// TIA Portal project "Traffic_feuxFBD" (V15)

(* hardware
DEVICE "Station S7300/ET200M_1"  S7-300 station
   slot 0: "Châssis_0"  Rail  6ES7 390-1***0-0AA0
   slot 2: "PLC_1"  CPU 315-2 PN/DP  6ES7 315-2EH14-0AB0  V3.2
      slot 2: "Interface PROFINET_1"  PN-IO
         slot 1: "Port_1"  Port
         slot 2: "Port_2"  Port
DEVICE "HMI_1"  KTP900 Basic PN
   slot 0: "HMI_1"  KTP900 Basic PN  6AV2 123-2JB03-0AX0  15.0.0.0
   slot 1: "HMI_RT_1"  KTP900 Basic PN  6AV2 123-2JB03-0AX0  15.0.0.0
   slot 5: "HMI_1.IE_CP_1"  PROFINET Interface  15.0.0.0
      slot 1: "Interface PROFINET_1"  PROFINET Interface
         slot 1: "Port_1"  Port
*)

// ===== PLC "PLC_1"  CPU 315-2 PN/DP =====

VAR_GLOBAL   // PLC tag table "Light_table"
   "Lred" AT %Q0.0 : Bool;
   "Lgreen" AT %Q0.1 : Bool;
   "Lorange" AT %Q0.2 : Bool;
   "Start" AT %I0.0 : Bool;
END_VAR

DATA_BLOCK "Bloc_1_DB"   // DB1
{ S7_Optimized_Access := 'FALSE' }
VERSION : 0.1
// stored: InstanceOfName Bloc_1
"Bloc_1"
BEGIN
END_DATA_BLOCK

FUNCTION_BLOCK "Bloc_1"   // FB1, GRAPH
{ S7_Optimized_Access := 'FALSE' }
VERSION : 0.1
   VAR_INPUT
      OFF_SQ : Bool := false;   // Désactiver le graphe
      INIT_SQ : Bool := false;   // Mettre le graphe à l'état initial
      ACK_EF : Bool := false;   // Acquitter toutes les erreurs et perturbations
      S_PREV : Bool := false;   // Afficher l'étape précédente dans le paramètre S_NO
      S_NEXT : Bool := false;   // Afficher l'étape suivante dans le paramètre S_NO
      SW_AUTO : Bool := false;   // Mode automatique
      SW_TAP : Bool := false;   // Mode semi-automatique/Activation de l'étape suivante avec transition
      SW_TOP : Bool := false;   // Mode semi-automatique/Ignorer la transition
      SW_MAN : Bool := false;   // Mode manuel
      S_SEL : Int := 0;   // Sélectionner l'étape à afficher dans S_NO
      S_ON : Bool := false;   // Activer l'étape figurant dans le paramètre S_NO
      S_OFF : Bool := false;   // Désactiver l'étape figurant dans le paramètre S_NO
      T_PUSH : Bool := false;   // Validation de commutation pour transition en mode semi-automatique
   END_VAR
   VAR_OUTPUT
      S_NO : Int := 0;   // Numéro d'étape
      S_MORE : Bool := false;   // Il existe d'autres étapes qui peuvent être affichées dans S_NO.
      S_ACTIVE : Bool := false;   // L'étape affichée dans le paramètre S_NO est activée
      ERR_FLT : Bool := false;   // Erreur groupée Interlock or Supervision
      AUTO_ON : Bool := false;   // Mode automatique activé
      TAP_ON : Bool := false;   // Mode semi-automatique/Etape avec transition activé
      TOP_ON : Bool := false;   // Mode semi-automatique/Ignorer la transition activé
      MAN_ON : Bool := false;   // Mode manuel activé
   END_VAR
   VAR
      SWITCH : Array[0..0] of DWord;
      SW_SQTS : Array[0..3] of Byte;
      SW_ADDR : Word := 16#A;
      G7T_0 : GraphTransition;
      G7S_0 : GraphStep;
      PRE_CRIT : Array[0..0] of DWord;
      POST_CRIT : Array[0..0] of DWord;
      TVX : Array[0..2] of Byte;
      TTX : Array[0..2] of Byte;
      TSX : Array[0..2] of Byte;
      S00X : Array[0..2] of Byte;
      SOFFX : Array[0..2] of Byte;
      SONX : Array[0..2] of Byte;
      SAX : Array[0..2] of Byte;
      SERRX : Array[0..4] of Byte;
      SMX : Array[0..4] of Byte;
      S0X : Array[0..4] of Byte;
      S1X : Array[0..4] of Byte;
      S_DISPLAY : Int;   // Affichage interne du paramètre de sortie S_NO
      S_SEL_OLD : Int;   // Valeur précédente dans S_SEL
      S_DISPIDX : Byte;   // Indice de l'étape affichée dans S_NO
      T_DISPIDX : Byte;   // Indice de la transition affichée dans T_NO
      MOPEDGE : Struct
         AUTO : Bool := false;
         MAN : Bool := false;
         TAP : Bool := false;
         TOP : Bool := false;
         ACK_S : Bool := false;
         REG_S : Bool := false;
         T_PREV : Bool := false;
         T_NEXT : Bool := false;
         LOCK : Bool := false;
         SUP : Bool := false;
         ACKREQ : Bool := false;
         SSKIP : Bool := false;
         OFF : Bool := false;
         INIT : Bool := false;
         HALT : Bool := false;
         TMS_HALT : Bool := false;
         OPS_ZERO : Bool := false;
         SACT_DISP : Bool := false;
         SEF_DISP : Bool := false;
         SALL_DISP : Bool := false;
         S_PREV : Bool := false;
         S_NEXT : Bool := false;
         S_SELOK : Bool := false;
         S_ON : Bool := false;
         S_OFF : Bool := false;
         T_PUSH : Bool := false;
         REG : Bool := false;
         ACK : Bool := false;
         IL_PERM : Bool := false;
         T_PERM : Bool := false;
         ILP_MAN : Bool := false;
      END_STRUCT;
      MOP : Struct   // Mode de fonctionnement
         AUTO : Bool := true;   // Etat : Mode automatique
         MAN : Bool := false;   // Etat : Mode manuel
         TAP : Bool := false;   // Etat : Mode semi-automatique/Activation de l'étape suivante avec transition
         TOP : Bool := false;   // Etat : Mode semi-automatique/Ignorer la transition
         ACK_S : Bool := false;   // Requête : Acquitter l'étape figurant dans le paramètre S_NO
         REG_S : Bool := false;   // Requête : Enregistrer l'étape figurant dans le paramètre S_NO
         T_PREV : Bool := false;   // Requête : Afficher la transition valide précédente dans le paramètre T_NO
         T_NEXT : Bool := false;   // Requête : Afficher la transition valide suivante dans le paramètre T_NO
         LOCK : Bool := true;   // Etat : Traitement des Interlocks activé
         SUP : Bool := true;   // Etat : Traitement de Supervision activé
         ACKREQ : Bool := true;   // Etat : Acquittement requis
         SSKIP : Bool := false;   // Etat : "Ignorer les étapes" activé
         OFF : Bool := false;   // Requête : Désactiver toutes les étapes
         INIT : Bool := true;   // Requête : Mettre le graphe à l'état initial
         HALT : Bool := false;   // Etat : Le graphe est arrêté
         TMS_HALT : Bool := false;   // Etat : Toutes les temporisations internes sont arrêtées
         OPS_ZERO : Bool := false;   // Etat : Tous les opérandes traités avec N, L, D mis à 0
         SACT_DISP : Bool := true;   // Etat : N'afficher que les étapes actives
         SEF_DISP : Bool := false;   // Etat : Afficher uniquement les étapes avec erreurs et perturbations
         SALL_DISP : Bool := false;   // Etat : Afficher toutes les étapes
         S_PREV : Bool := false;   // Requête : Afficher l'étape précédente dans le paramètre S_NO
         S_NEXT : Bool := false;   // Requête : Afficher l'étape suivante dans le paramètre S_NO
         S_SELOK : Bool := false;   // Requête : Afficher dans le paramètre S_NO le numéro d'étape figurant dans S_SEL
         S_ON : Bool := false;   // Requête : Activer l'étape figurant dans le paramètre S_NO
         S_OFF : Bool := false;   // Requête : Désactiver l'étape figurant dans le paramètre S_NO
         T_PUSH : Bool := false;   // Requête : Validation de commutation pour transition
         REG : Bool := false;   // Requête : Enregistrer toutes les erreurs Interlock et Supervision
         ACK : Bool := false;   // Requête : Acquitter toutes les erreurs Interlock et Supervision
         IL_PERM : Bool := false;   // Etat : Traitement permanent de tous les Interlocks
         T_PERM : Bool := false;   // Etat : Traitement permanent de toutes les transitions
         ILP_MAN : Bool := false;   // Etat : Traitement permanent de tous les Interlocks en mode manuel
      END_STRUCT;
      TICKS : Struct   // Périodes d'horloge
         DELTA : Time := T#0ms;   // Différence de temps entre deux cycles
         OLD : Time := T#0ms;   // Valeur du compteur de périodes 10 ms au dernier cycle
         NEW : Time := T#0ms;   // Valeur du compteur de périodes 10 ms dans ce cycle
      END_STRUCT;
      SQ_FLAGS : Struct   // Mémentos de graphe
         ERR_FLT : Bool := false;   // Erreur groupée Interlock et Supervision
         ERROR : Bool := false;   // Erreur groupée Interlock
         FAULT : Bool := false;   // Erreur groupée Supervision
         RT_FAIL : Bool := false;   // Erreur à l'exécution
         NO_SNO : Bool := false;   // Numéro d'étape requis introuvable
         NF_OFL : Bool := false;   // Débordement : Trop de requêtes ON ou OFF
         SA_OFL : Bool := false;   // Débordement : Trop d'étapes activées
         TV_OFL : Bool := false;   // Débordement : Trop de transitions valides
         MSG_OFL : Bool := false;   // Débordement : Pas assez de ressources système pour ALARM_S
         NO_SWI : Bool := false;   // Pas de commutation dans ce cycle
         CYC_OP : Bool := false;   // Exécution cyclique du graphe après l'initialisation
         AS_MSG : Bool := true;   // Messages à l'exécution activés ou désactivés par instruction
         AS_SEND : Bool := false;   // Envoyer les messages de WR_USMSG ou les entrer uniquement dans le tampon de diagnostic
         SQ_BUSY : Bool := false;   // Mémento de front interne pour le traitement séquentiel
         SA_BUSY : Bool := false;   // Mémento de front interne pour le traitement séquentiel
         AS_SIG : Bool := false;   // Mémentos de front pour messages de Alarm_S et Alarm_SQ
      END_STRUCT;
      S_PTR : DWord := 16#2A0;
      S_PTR2 : DWord := 16#0;
      S_PTR3 : DWord := 16#850;
      S_PTR4 : DWord := 16#820;
      T_PTR : DWord := 16#7F0;
      C_AR2 : DWord := 16#0;
      M_FBDB : DWord := 16#10000;
      M_SNO : Word := 16#0;
      M_EVID : Word := 16#0;
      M_EVIL : C_Alarm_s;
      M_EVSV : C_Alarm_s;
      M_EV : DWord := 16#760;
      CRIT : Array[0..31] of Bool;
      S_START : Byte := 16#0;
      S_IDX : Byte := 16#0;
      S_INT : Int := 72;
      S_TMP : Byte := 16#0;
      T_START : Byte := 16#0;
      T_IDX : Byte := 16#0;
      T_TMP : Byte := 16#0;
      T_TMP2 : Byte := 16#00;
      TV_POT : Byte := 16#06;
      RETURN1 : Byte := 16#0;
      RETURN2 : Byte := 16#0;
      SINI : Array[0..2] of Byte;
      LSTT : Array[0..3] of Byte;
      ATAJ : Array[0..3] of Byte;
      ATAB : Array[0..3] of Byte;
      PSTT : Array[0..3] of Byte;
      NSTT : Array[0..3] of Byte;
      ASSJ : Array[0..3] of Byte;
      ASSB : Array[0..3] of Byte;
      PTTS : Array[0..3] of Byte;
      NTTS : Array[0..3] of Byte;
      PRE_CNT : Word := 16#1;
      POST_CNT : Word := 16#1;
      ADR_COND : Word := 16#0;
      MAX_TVAL : Byte := 16#1;
      MAX_SACT : Byte := 16#1;
      MAX_CRIT : Byte := 16#4;
      T_CNT : Byte := 16#3;
      SUP_CNT : Byte := 16#0;
      LOCK_CNT : Byte := 16#0;
      S_CNT : Byte := 16#3;
      SQ_CNT : Byte := 16#1;
      PRS_INPAR : DWord := 16#E000FEC8;
      PRS_OUTPAR : DWord := 16#E000800F;
      GC_FLAGS : Struct
         T_MACH : Byte := 16#EB;
         COND_ED : Byte := 16#E3;
         W_LEVEL : Byte := 16#D5;
         FB_IF : Byte := 16#FA;
         AS_MSG : Word := 16#404;
         SSB : Word := 16#108;
         DILG : Word := 16#1B8;
         ADDR_T0 : Word := 16#14;
         CRIT_AVAIL : Bool := false;
         SSKIP_AVAIL : Bool := true;
         SSKIP_ON : Bool := false;
         ACK_REQ : Bool := true;
         SYNC_AVAIL : Bool := true;
         ILP_MAN : Bool := false;
         SWM_LOCKED : Bool := false;
         SAVE_SW : Bool := true;
      END_STRUCT;
      G7_FBMARK : Byte := 16#3C;
      G7_RELEASE : Byte := 16#3C;
      G7_ID2 : Byte := 16#37;
      G7_ID1 : Byte := 16#47;
   END_VAR
   // SW_SQTS[0] := 16#1;
   // TVX[0] := 16#1;
   // TTX[0] := 16#1;
   // TSX[0] := 16#1;
   // S00X[0] := 16#1;
   // SOFFX[0] := 16#1;
   // SONX[0] := 16#1;
   // SAX[0] := 16#1;
   // SERRX[0] := 16#1;
   // SMX[0] := 16#1;
   // S0X[0] := 16#1;
   // S1X[0] := 16#1;
   // SINI[0] := 16#2;
   // SINI[1] := 16#1;
   // SINI[2] := 0;
   // LSTT[0] := 0;
   // LSTT[1] := 0;
   // LSTT[2] := 0;
   // LSTT[3] := 16#1;
   // ATAJ[0] := 0;
   // ATAJ[1] := 16#1;
   // ATAJ[2] := 16#2;
   // ATAJ[3] := 16#3;
   // ATAB[0] := 0;
   // ATAB[1] := 16#1;
   // ATAB[2] := 16#2;
   // ATAB[3] := 16#3;
   // PSTT[0] := 0;
   // PSTT[1] := 16#1;
   // PSTT[2] := 16#2;
   // PSTT[3] := 16#3;
   // NSTT[0] := 16#1;
   // NSTT[1] := 16#2;
   // NSTT[2] := 16#3;
   // NSTT[3] := 16#1;
   // ASSJ[0] := 0;
   // ASSJ[1] := 16#1;
   // ASSJ[2] := 16#2;
   // ASSJ[3] := 16#3;
   // ASSB[0] := 0;
   // ASSB[1] := 16#1;
   // ASSB[2] := 16#2;
   // ASSB[3] := 16#3;
   // PTTS[0] := 0;
   // PTTS[2] := 16#1;
   // PTTS[3] := 16#2;
   // NTTS[0] := 0;
   // NTTS[1] := 16#1;
   // NTTS[2] := 16#2;
   // NTTS[3] := 16#3;
BEGIN
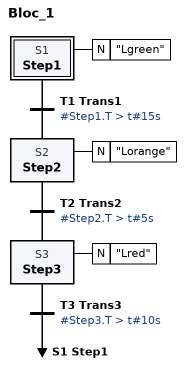
   // sequencer 1
   INITIAL_STEP Step1:   // S1
              N    "Lgreen"
   END_STEP
   TRANSITION Trans1 FROM Step1 TO Step2   // T1
      := #Step1.T > t#15s;
   END_TRANSITION
   STEP Step2:   // S2
              N    "Lorange"
   END_STEP
   TRANSITION Trans2 FROM Step2 TO Step3   // T2
      := #Step2.T > t#5s;
   END_TRANSITION
   STEP Step3:   // S3
              N    "Lred"
   END_STEP
   TRANSITION Trans3 FROM Step3 TO Step1   // T3, jump
      := #Step3.T > t#10s;
   END_TRANSITION
END_FUNCTION_BLOCK

ORGANIZATION_BLOCK "Main"   // OB1, LAD
TITLE = "Main Program Sweep (Cycle)"
{ S7_Optimized_Access := 'FALSE' }
VERSION : 0.1
   VAR_TEMP
      OB1_EV_CLASS : Byte;   // Bits 0-3 = 1 (Coming event), Bits 4-7 = 1 (Event class 1)
      OB1_SCAN_1 : Byte;   // 1 (Cold restart scan 1 of OB 1), 3 (Scan 2-n of OB 1)
      OB1_PRIORITY : Byte;   // Priority of OB Execution
      OB1_OB_NUMBR : Byte;   // 1 (Organization block 1, OB1)
      OB1_RESERVED_1 : Byte;   // Reserved for system
      OB1_RESERVED_2 : Byte;   // Reserved for system
      OB1_PREV_CYCLE : Int;   // Cycle time of previous OB1 scan (milliseconds)
      OB1_MIN_CYCLE : Int;   // Minimum cycle time of OB1 (milliseconds)
      OB1_MAX_CYCLE : Int;   // Maximum cycle time of OB1 (milliseconds)
      OB1_DATE_TIME : Date_And_Time;   // Date and time OB1 started
   END_VAR
BEGIN

REGION Network 1
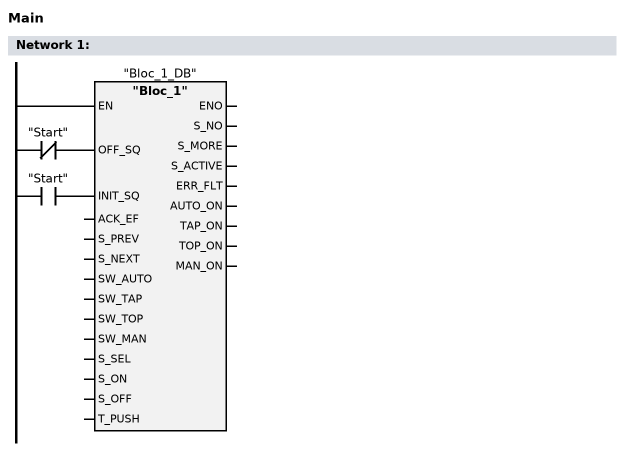
   RUNG wire#powerrail
      "Bloc_1_DB"(OFF_SQ := wire#w1, INIT_SQ := wire#w2, ACK_EF :=, S_PREV :=, S_NEXT :=, SW_AUTO :=, SW_TAP :=, SW_TOP :=, SW_MAN :=, S_SEL :=, S_ON :=, S_OFF :=, T_PUSH :=, S_NO =>, S_MORE =>, S_ACTIVE =>, ERR_FLT =>, AUTO_ON =>, TAP_ON =>, TOP_ON =>, MAN_ON =>)
   END_RUNG
   RUNG wire#powerrail
      I_Contact( "Start" )
   END_RUNG wire#w1
   RUNG wire#powerrail
      Contact( "Start" )
   END_RUNG wire#w2
   // the same network as SCL:
   "Bloc_1_DB"(OFF_SQ := NOT "Start", INIT_SQ := "Start");   // "Bloc_1"
END_REGION
END_ORGANIZATION_BLOCK

(* ===== HMI "HMI_RT_1" =====
system functions are stored by id; their names below are inferred from use
connection "HMI_Liaison_1": ETHERNET, SIMATIC S7 300/400 MPI

HMI tags "Table de variables standard"
   "Numéro_vue_variable" : UInt, internal
   "Lgreen" : Bool = PLC Lgreen AT %Q0.1, 1 s
   "Lorange" : Bool = PLC Lorange AT %Q0.2, 1 s
   "Lred" : Bool = PLC Lred AT %Q0.0, 1 s
   "Start" : Bool = PLC Start AT %I0.0, 1 s

text list "Nom_vue_liste_textes": 1 'Vue racine'

screen "Vue racine" 800x480, template "Modèle_1"
   on GenerateScreen: SetTag("Numéro_vue_variable", 1)
   Circle "Cercle_1" at 314,93 size 48x48
      Appearance <- "Lgreen"
   Circle "Cercle_2" at 314,141 size 48x48
      Appearance <- "Lorange"
   Circle "Cercle_3" at 314,187 size 48x48
      Appearance <- "Lred"
   Button "Bouton_1" at 49,111 size 78x27; TextOff 'Start'
      on Press: SetBit("Start")
   Button "Bouton_2" at 49,147 size 80x31; TextOff 'stop'
      on Press: ResetBit("Start")
   GraphicView "Vue de graphique_1" at 314,229 size 49x69; Picture "Graphique_1"
   TextField "Champ de texte_1" at 248,53 size 126x28; Text 'Traffic_Light'

Template "Modèle_1" 800x480
   SymbolicIOField "Vue_champ_ES_symbolique" at 2,7 size 691x26; TextOff '0'; TextOn '1'; TextList "Nom_vue_liste_textes"
      ProcessValue <- "Numéro_vue_variable"
      on Change: ActivateScreenByNumber("Numéro_vue_variable", 0)
   DateTimeField "HmiScreenItemData" at 695,20 size 105x20
   DateTimeField "HmiScreenItemData_1" at 695,0 size 105x20
*)